{attribute 'GeneratedUsingTerminal: EJ9404-0000-0000'}
{attribute addProperty BoxType "EJ9404-0000-0000"}
{attribute addProperty Description "EJ9404-0000 Power supply module 12A"}
{attribute addProperty Physics "KK"}
{attribute addProperty Id "EJ9404"}
{attribute addProperty CRC "2785896704"}
{attribute addProperty Size "0"}
TYPE EJ9404_A60D6900 EXTENDS EtcSlaveTerminalBase_947E5A46 :
STRUCT
END_STRUCT
END_TYPE

(* stored: Version 1.2.0.0, ProductVersion 3.1.4024.11
   DUT EJ9404_A60D6900: Id {95978cd6-5934-474f-ad9b-f4b78b9ac497} *)
